// Mitsubishi GX Works2 project: 0624(상승_하강펄스)   PLC: Q02/Q02H

PROGRAM MAIN
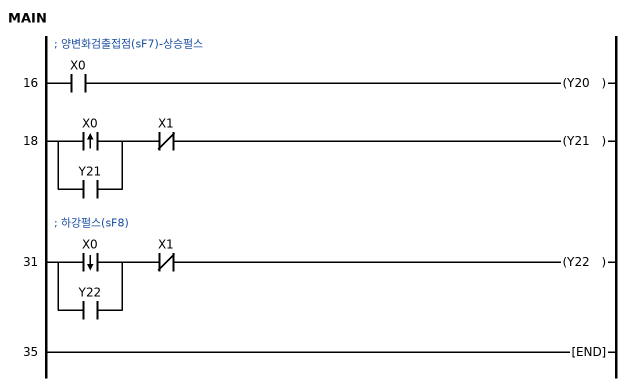
; 양변화검출접점(sF7)-상승펄스
16    LD      X0
      OUT     Y20
18    LDP     X0
      OR      Y21
      ANI     X1
      OUT     Y21
; 하강펄스(sF8)
31    LDF     X0
      OR      Y22
      ANI     X1
      OUT     Y22
35    END
END_PROGRAM
